(* IEC 61131-3 sources: stc/cmd/stc/testdata, 3 files *)

(* ---- emit_oop.st ---- *)
FUNCTION_BLOCK MyFB
VAR
    counter : INT;
END_VAR
    counter := counter + 1;

METHOD PUBLIC DoWork : BOOL
VAR_INPUT
    value : INT;
END_VAR
    DoWork := value > 0;
END_METHOD

END_FUNCTION_BLOCK

(* ---- emit_simple.st ---- *)
PROGRAM Main
VAR
    x : INT;
    y : REAL;
END_VAR
    x := 42;
    y := 3.14;
END_PROGRAM

(* ---- sim_test.st ---- *)
PROGRAM SimTest
VAR_INPUT
    SENSOR : REAL;
END_VAR
VAR_OUTPUT
    OUTPUT : REAL;
END_VAR
    OUTPUT := SENSOR * 2.0;
END_PROGRAM
